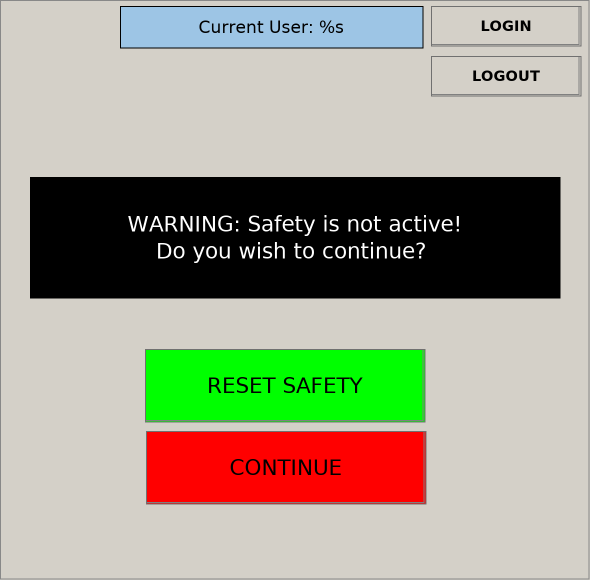
VISUALIZATION safetyDisableWarning  // 590x580
    Rectangle (30,177 530x121), "WARNING: Safety is not active! Do you wish to continue?", text variable: MAIN.sSafetyResetMsg
    Button (145,349 280x73), "RESET SAFETY"
        toggle GVL_machine.bSafetyBypass
    Button (146,431 280x73), "CONTINUE"
        OnMouseDown: change screen: Previous 
        OnMouseDown: execute { main.fbSafetyBypassTim(IN := FALSE); }
    Button (431,6 150x40), "LOGIN"
        OnMouseDown: VisuUserMgmt Type=Login
    Button (431,56 150x40), "LOGOUT"
        OnMouseDown: VisuUserMgmt Type=Logout
    Textfield (120,6 303x42), "Current User: %s", text variable: VisuElems.CurrentUserName
END_VISUALIZATION

(* stored: Version 1.1.0.1, ProductVersion 3.1.4024.13
   Visu safetyDisableWarning: Id {e10ce054-e718-4f7a-9e60-2f79bef52ca3} *)
